ABB RAPID module: Socket_Server.mod

MODULE Module2
    ! The socket communication and other variables.
	VAR socketdev server_socket;
	VAR socketdev client_socket;
	VAR string recv_string1;
	VAR string recv_string2;
	VAR string recv_string3;
	VAR string recv_string4;
	VAR robtarget to_point;
	VAR jointtarget to_joint_pos;
	VAR bool keep_scanning;
    VAR bool filler_bool;

    VAR confdata conf := [0,0,0,0];
    PERS tooldata T_TEXT_01:=[TRUE,[[-90.442,-25.934,132.491],[0.77729,-0.25919,-0.06870,0.56914]],[3.000,[-90.442,-25.934,132.491],[1,0,0,0],0,0,0]];
    TASK PERS wobjdata DefaultFrame:=[FALSE,TRUE,"",[[0.000,0.000,0.000],[1.00000,0.00000,0.00000,0.00000]],[[0,0,0],[1,0,0,0]]];
    TASK PERS speeddata Speed000:=[200.000,180.000,5000.000,1080.000];
    TASK PERS speeddata Speed001:=[20.000,180.000,5000.000,1080.000];
    TASK PERS zonedata Zone000:=[FALSE,1.000,1.000,1.000,0.100,1.000,0.100];
    TASK PERS zonedata Zone001:=[FALSE,1.000,1.000,1.000,0.100,1.000,0.100];

    VAR speeddata current_speed;

    PROC main()
        ! Close any leftover sockets.
		SocketClose client_socket;
		SocketClose server_socket;

        SocketCreate server_socket;
		SocketBind server_socket, "127.0.0.1", 1025;
		SocketListen server_socket;
		SocketAccept server_socket, client_socket \Time:=WAIT_MAX;

        keep_scanning := TRUE;
        recv_string1 := ClientSync();

        IF(recv_string1 = "ok") THEN
            WHILE keep_scanning DO

                !recv_string1 := ClientSync();
                SocketReceive client_socket \Str:=recv_string2 \Time:=3;
                SocketReceive client_socket \Str:=recv_string3 \Time:=3;
                SocketReceive client_socket \Str:=recv_string4 \Time:=3;

                IF recv_string4 = "Speed000" THEN
                    current_speed := Speed000;
                ELSEIF recv_string4 = "Speed001" THEN
                    current_speed := Speed001;
                ENDIF

                IF recv_string2 = "MoveL" THEN
                     filler_bool:= StrToVal(recv_string3, to_point);
                     MoveL to_point,current_speed,Zone001,T_TEXT_01 \WObj:=DefaultFrame;
                ELSEIF recv_string2 = "MoveAbsJ" THEN
                    filler_bool:= StrToVal(recv_string3, to_joint_pos);
                    MoveAbsJ to_joint_pos,current_speed,Zone000,T_TEXT_01;
                ENDIF
                WaitTime \InPos,0;
                SocketSend client_socket \Str:="ready";
            ENDWHILE
        ENDIF
        !ERROR
           ! IF ERRNO=ERR_SOCK_TIMEOUT THEN
               ! keep_scanning := FALSE;
                !RETURN;
            !ENDIF
    ENDPROC

	! Wait until the client sends a string.
	FUNC string ClientSync()
		VAR string recv_string;
		SocketReceive client_socket \Str:=recv_string \Time:=WAIT_MAX;
		IF recv_string = "listening?" THEN
			SocketSend client_socket \Str:="Yes";
			RETURN "ok";
		ELSEIF recv_string = "stop" THEN
			SocketSend client_socket \Str:="ok";
			RETURN "stop";
		ELSE
            !switching protocols

			RETURN "unexpect str:";
		ENDIF
	ENDFUNC

    FUNC string GetTargets()
        VAR string recv_string;
        SocketReceive client_socket \Str:=recv_string \Time:=WAIT_MAX;
    ENDFUNC
ENDMODULE
